// TIA Portal V16 export
// export: Created 2021-08-04T23:04:17.8933122Z, ExportSetting WithDefaults, DisplayName Totally Integrated Automation Portal, DisplayVersion V16 Update 4, DisplayName TIA Portal Version Control Interface, DisplayVersion V16 Update 2, DisplayName TIA Portal Openness, DisplayVersion V16 Update 4, DisplayName STEP 7 Professional, DisplayVersion V16 Update 4, DisplayName STEP 7 Safety, DisplayVersion V16, DisplayName WinCC Advanced, DisplayVersion V16 Update 4
FUNCTION_BLOCK "Main_Safety_RTG1"   // FB1, F_FBD
{ S7_Optimized_Access := 'TRUE' }
VERSION : 0.1
// stored: AutoNumber false, IsIECCheckEnabled false, UDAEnableTagReadback false
BEGIN

REGION Network 1
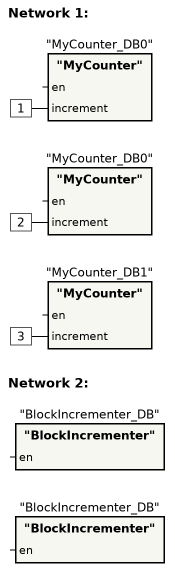
   "MyCounter_DB0"(increment := 1);   // "MyCounter"
   "MyCounter_DB0"(increment := 2);   // "MyCounter"
   "MyCounter_DB1"(increment := 3);   // "MyCounter"
END_REGION

REGION Network 2
   "BlockIncrementer_DB"();   // "BlockIncrementer"
   "BlockIncrementer_DB"();   // "BlockIncrementer"
END_REGION
END_FUNCTION_BLOCK
